FUNCTION SPLITTING_WORD_INTO_BOOLS
  (* Standard: 61499-1; Description: Copyright (c) 2024 HR Agrartechnik GmbH This program and the accompanying materials are made available under the terms of the Eclipse Public License 2.0 which is available at https://www.eclipse.org/legal/epl-2.0/ SPDX-License-Identifier: EPL-2.0 *)
  (* Version 1.0, 2024-02-22, franz *)
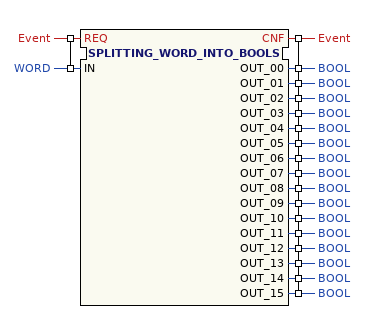
  EVENT_INPUT
    REQ WITH IN; (* Normal Execution Request *)
  END_EVENT
  EVENT_OUTPUT
    CNF WITH OUT_00, OUT_01, OUT_02, OUT_03, OUT_04, OUT_05, OUT_06, OUT_07, OUT_08, OUT_09, OUT_10, OUT_11, OUT_12, OUT_13, OUT_14, OUT_15; (* Execution Confirmation *)
  END_EVENT
  VAR_INPUT
    IN : WORD; (* WORD Input *)
  END_VAR
  VAR_OUTPUT
    OUT_00 : BOOL; (* BIT 00 *)
    OUT_01 : BOOL; (* BIT 01 *)
    OUT_02 : BOOL; (* BIT 02 *)
    OUT_03 : BOOL; (* BIT 03 *)
    OUT_04 : BOOL; (* BIT 04 *)
    OUT_05 : BOOL; (* BIT 05 *)
    OUT_06 : BOOL; (* BIT 06 *)
    OUT_07 : BOOL; (* BIT 07 *)
    OUT_08 : BOOL; (* BIT 08 *)
    OUT_09 : BOOL; (* BIT 09 *)
    OUT_10 : BOOL; (* BIT 10 *)
    OUT_11 : BOOL; (* BIT 11 *)
    OUT_12 : BOOL; (* BIT 12 *)
    OUT_13 : BOOL; (* BIT 13 *)
    OUT_14 : BOOL; (* BIT 14 *)
    OUT_15 : BOOL; (* BIT 15 *)
  END_VAR
  BODY IN ST:
FUNCTION SPLITTING_WORD_INTO_BOOLS

VAR_INPUT
	IN : WORD;    // WORD Input
END_VAR

VAR_OUTPUT
	OUT_00 : BOOL;    // BIT 00
	OUT_01 : BOOL;    // BIT 01
	OUT_02 : BOOL;    // BIT 02
	OUT_03 : BOOL;    // BIT 03
	OUT_04 : BOOL;    // BIT 04
	OUT_05 : BOOL;    // BIT 05
	OUT_06 : BOOL;    // BIT 06
	OUT_07 : BOOL;    // BIT 07
	OUT_08 : BOOL;    // BIT 08
	OUT_09 : BOOL;    // BIT 09
	OUT_10 : BOOL;    // BIT 10
	OUT_11 : BOOL;    // BIT 11
	OUT_12 : BOOL;    // BIT 12
	OUT_13 : BOOL;    // BIT 13
	OUT_14 : BOOL;    // BIT 14
	OUT_15 : BOOL;    // BIT 15
END_VAR

(* this Function extracts the 16 BOOLS from a word *)
OUT_00 := IN.0;
OUT_01 := IN.1;
OUT_02 := IN.2;
OUT_03 := IN.3;
OUT_04 := IN.4;
OUT_05 := IN.5;
OUT_06 := IN.6;
OUT_07 := IN.7;
OUT_08 := IN.8;
OUT_09 := IN.9;
OUT_10 := IN.10;
OUT_11 := IN.11;
OUT_12 := IN.12;
OUT_13 := IN.13;
OUT_14 := IN.14;
OUT_15 := IN.15;

END_FUNCTION
  END_BODY
END_FUNCTION
